// TIA Portal V20 export
TYPE "typeIdentRfHmi"
// stored: Access Published
   STRUCT
      selectedUnit : USInt;
      selectedEM : USInt;
      rfReaderId : USInt;   // Reader ID / RF Reader ID
      numberOfRf : USInt;   // Anzahl der RFID Antriebe / Number of used RFIDs
      rfReader : Array[0.."NO_OF_RF_IDENT_DEVICES"] of "LSicar_typeIdentInterfaceHmi";   // RF Reader
   END_STRUCT;
END_TYPE
